{attribute addProperty BoxType "EL6692-0002-0016"}
{attribute addProperty Id "SYNC_InputsAT %I*SYNC_Inputs_AD8FC9014860IO_InputsEMPTY_STRUCTURE000IO_OutputsEMPTY_STRUCTURE000WcStateAT %I*WcState_F855686C1620InfoDataAT %I*InfoData_275E3363128160"}
{attribute addProperty CRC "3781676361"}
{attribute addProperty SizeInBites "192"}
{attribute addProperty SizeInBytes "24"}
TYPE EL6692_9D416E6E :
STRUCT
	{attribute addProperty Name "SYNC_Inputs"}
	SYNC_Inputs : SYNC_Inputs_AD8FC901;
	{attribute addProperty Name "IO_Inputs"}
	IO_Inputs : EMPTY_STRUCTURE;
	{attribute addProperty Name "IO_Outputs"}
	IO_Outputs : EMPTY_STRUCTURE;
	{attribute addProperty Name "WcState"}
	WcState : WcState_F855686C;
	{attribute addProperty Name "InfoData"}
	InfoData : InfoData_275E3363;
END_STRUCT
END_TYPE

(* stored: Version 1.2.0.0, ProductVersion 3.1.4024.9
   DUT EL6692_9D416E6E: Id {8a865f40-27e7-4c75-8255-b38792204ae5} *)
